// TIA Portal V20 export
DATA_BLOCK "progalarme_DB"   // DB6
// stored: InstanceOfName progalarme, InstanceOfType FB
"progalarme"
   // VAR_INPUT
   //    AlarmInput : Bool;
   //    AlarmText : String;
   //    Tag : String;
   // END_VAR
   // VAR_IN_OUT
   //    Program_Alarm_1 : Program_Alarm;
   // END_VAR
   // VAR
   //    Program_Alarm_2 { S7_SetPoint := 'True'} : Program_Alarm;
   // END_VAR
BEGIN
END_DATA_BLOCK
